FUNCTION_BLOCK Basic (* Basic FB with empty ECC *)
  (* Standard: 61499-2 *)
  (* Version 1.0, 2016-05-26, AZ, fortiss GmbH *)
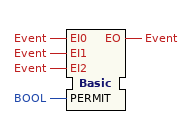
  EVENT_INPUT
    EI0;
    EI1;
    EI2;
  END_EVENT
  EVENT_OUTPUT
    EO;
  END_EVENT
  VAR_INPUT
    PERMIT : BOOL;
  END_VAR
  EC_STATES
    START; (* Initial State *)
  END_STATES
END_FUNCTION_BLOCK
